// TwinCAT 3 PLC project PLC
// ProgramVersion: 3.1.4024.0
// libraries:
//   Tc2_Standard, * (Beckhoff Automation GmbH)
//   Tc2_System, * (Beckhoff Automation GmbH)
//   Tc3_IotBase, * (Beckhoff Automation GmbH)
//   Tc3_Module, * (Beckhoff Automation GmbH)
// project tree:
//   DUTs/ sProcessData.TcDUT
//   GVLs/ GVL.TcGVL
//   / PlcTask.TcTTO
//   POUs/ MAIN.TcPOU, PRG_MQTT_Client.TcPOU, PRG_ProcessSimulation.TcPOU
// real-time tasks:
//   TASK PlcTask: cycle T#10ms, priority 20, ADS port 350

CONFIGURATION PLC
    RESOURCE PLC ON TwinCAT3
        TASK PlcTask(INTERVAL := T#10ms, PRIORITY := 20);
        PROGRAM MAIN WITH PlcTask : MAIN;
    END_RESOURCE
END_CONFIGURATION

// ---- DUTs/sProcessData.TcDUT
TYPE sProcessData :
STRUCT
	rTemperature : REAL;
    rPressure : REAL;
    rFlowRate : REAL;
END_STRUCT
END_TYPE

// ---- GVLs/GVL.TcGVL
{attribute 'qualified_only'}
VAR_GLOBAL

	g_stProcessData : sProcessData;

	//Cycle Counter
	g_iCounter : INT := 0;
	
	//Control Button
	g_bStart : BOOL := FALSE;
    g_bStop  : BOOL := TRUE;
    g_bReset : BOOL := FALSE;
	g_bExit  : BOOL := FALSE;
END_VAR

// ---- POUs/MAIN.TcPOU
PROGRAM MAIN
VAR
END_VAR

PRG_ProcessSimulation();
PRG_MQTT_Client();

END_PROGRAM

// ---- POUs/PRG_ProcessSimulation.TcPOU
PROGRAM PRG_ProcessSimulation
VAR
    rTempDelta : REAL := 0.05;
    rFlowDelta : REAL := 0.1;
END_VAR

// RESET data
IF GVL.g_bReset THEN
    GVL.g_iCounter := 0;
    GVL.g_stProcessData.rTemperature := 20.0;
    GVL.g_stProcessData.rPressure := 1.0;
    GVL.g_stProcessData.rFlowRate := 0.0;
    GVL.g_bReset := FALSE;
END_IF

// simulation data when get START
IF GVL.g_bStart AND NOT GVL.g_bStop THEN

    GVL.g_stProcessData.rTemperature :=GVL.g_stProcessData.rTemperature + rTempDelta;

    GVL.g_stProcessData.rPressure := 1.0 + (GVL.g_iCounter) * 0.001;

    GVL.g_stProcessData.rFlowRate := GVL.g_stProcessData.rFlowRate + rFlowDelta;
END_IF

END_PROGRAM

// ---- POUs/PRG_MQTT_Client.TcPOU
PROGRAM PRG_MQTT_Client
VAR
    fbMqttClient   : FB_IotMqttClient;
    fbMessageQueue : FB_IotMqttMessageQueue;
    fbMessage      : FB_IotMqttMessage;

    bSetParams     : BOOL := TRUE;
    bSubscribed    : BOOL := FALSE;

    sTopicPub      : STRING(255) := 'factory/data';
    sTopicSub      : STRING(255) := 'factory/command';
    sPayloadPub    : STRING(255);
    sPayloadSub    : STRING(255);

    // string for building Payload
    s1, s2, s3, s4, s5, s6, s7, s8 : STRING(255);
	
    (* timer for periodic publish *)
    fbTimer          : TON := (PT := T#1S);

END_VAR

// Init
IF bSetParams THEN
    bSetParams := FALSE;

    fbMqttClient.sClientId := 'PLC_Beckhoff';
    fbMqttClient.sHostName := '127.0.0.1';   // broker MQTT
    fbMqttClient.nHostPort := 1883;
    fbMqttClient.ipMessageQueue := fbMessageQueue;
END_IF

	// Connection
fbMqttClient.Execute(bConnect := TRUE);

//Subscribe
IF fbMqttClient.bConnected AND NOT bSubscribed THEN
    bSubscribed := fbMqttClient.Subscribe(
        sTopic := sTopicSub,
        eQoS := TcIotMqttQos.AtMostOnceDelivery
    );
END_IF

// getting PayloadSub
IF fbMessageQueue.nQueuedMessages > 0 THEN
    IF fbMessageQueue.Dequeue(fbMessage := fbMessage) THEN
        fbMessage.GetTopic(pTopic := ADR(sTopicSub), nTopicSize := SIZEOF(sTopicSub));
        fbMessage.GetPayload(pPayload := ADR(sPayloadSub), nPayloadSize := SIZEOF(sPayloadSub), bSetNullTermination := TRUE);

        IF sPayloadSub = 'START' THEN
            GVL.g_bStart := TRUE;
            GVL.g_bStop  := FALSE;
            GVL.g_bExit  := FALSE;
        ELSIF sPayloadSub = 'STOP' THEN
            GVL.g_bStop  := TRUE;
            GVL.g_bStart := FALSE;
        ELSIF sPayloadSub = 'RESET' THEN
            GVL.g_iCounter := 0;
        ELSIF sPayloadSub = 'EXIT' THEN
            GVL.g_bExit  := TRUE;
            GVL.g_bStart := FALSE;
        END_IF
    END_IF
END_IF

//  When Start public PayloadPub each 1 sec.
IF GVL.g_bStart THEN
	fbTimer(IN := TRUE);
    IF fbTimer.Q THEN
		fbTimer(IN := FALSE);
		GVL.g_iCounter := GVL.g_iCounter + 1;
		s1 := CONCAT('{"counter":', TO_STRING(GVL.g_iCounter));
		s2 := CONCAT(s1, ',"time_ms":');
		s3 := CONCAT(s2, TIME_TO_STRING(TIME()));
		s4 := CONCAT(s3, ',"Temperature_C":');
		s5 := CONCAT(s4, TO_STRING(GVL.g_stProcessData.rTemperature));
		s6 := CONCAT(s5, ',"Pressure_bar":');
		s7 := CONCAT(s6, TO_STRING(GVL.g_stProcessData.rPressure));
		s8 := CONCAT(s7, ',"Flow_lpm":');
		sPayloadPub := CONCAT(s8, TO_STRING(GVL.g_stProcessData.rFlowRate));
		sPayloadPub := CONCAT(sPayloadPub, '}');
		
		fbMqttClient.Publish(
			sTopic := sTopicPub,
			pPayload := ADR(sPayloadPub),
			nPayloadSize := LEN(sPayloadPub),
			eQoS := TcIotMqttQos.AtMostOnceDelivery,
			bRetain := FALSE,
			bQueue := FALSE
			);
	END_IF	
END_IF

END_PROGRAM
